// TIA Portal V21 export
DATA_BLOCK "GlobalData"   // DB5
{ S7_Optimized_Access := 'TRUE' }
// stored: MemoryReserve 100
   VAR
      restart : Bool;
   END_VAR
BEGIN
END_DATA_BLOCK
